TYPE "Processing_ShW"
VERSION : 0.1
   STRUCT
      Trigger : Bool;
   END_STRUCT;

END_TYPE

